# B&R Automation Studio project BottlePlant2 (part 2)

#### Main.st
```iecst
PROGRAM _INIT
	(* Insert code here *)
	gCamSequencer.Ctrl.MpAxisCamSequencer_0.Enable:=TRUE;
	gCamSequencer.Ctrl.MpAxisCamSequencer_1.Enable:=TRUE;
	gCamSequencer.State:=STATE_WORK_SEQUENCER;

	(* Zdefiniowanie podstawowych parametrów sequencera *)
	gCamSequencer.Ctrl.MpAxisCamSequencerPar_0.Deceleration:=1000;
	gCamSequencer.Ctrl.MpAxisCamSequencerPar_0.Configuration.Master:=ADR(gTranAxis);
	gCamSequencer.Ctrl.MpAxisCamSequencerPar_0.Configuration.StartState:=0;
	gCamSequencer.Ctrl.MpAxisCamSequencerPar_0.Configuration.State[0].Event[0].Type:=ncSIGNAL1;
	gCamSequencer.Ctrl.MpAxisCamSequencerPar_0.Configuration.State[0].Event[0].Attribute:=ncAT_ONCE;
	gCamSequencer.Ctrl.MpAxisCamSequencerPar_0.Configuration.State[0].Event[0].NextState:=1;

	gCamSequencer.Ctrl.MpAxisCamSequencerPar_0.Configuration.State[1].CompMode:=ncOFF;
	gCamSequencer.Ctrl.MpAxisCamSequencerPar_0.Configuration.State[1].CamProfileIndex:=16#ffff;
	gCamSequencer.Ctrl.MpAxisCamSequencerPar_0.Configuration.State[1].MasterCompDistance:=0;
	gCamSequencer.Ctrl.MpAxisCamSequencerPar_0.Configuration.State[1].SlaveCompDistance:=0;
	gCamSequencer.Ctrl.MpAxisCamSequencerPar_0.Configuration.State[1].MasterFactor:=400*100;
	gCamSequencer.Ctrl.MpAxisCamSequencerPar_0.Configuration.State[1].SlaveFactor:=400*100;
	gCamSequencer.Ctrl.MpAxisCamSequencerPar_0.Configuration.State[1].Event[0].Type:=ncST_END;
	gCamSequencer.Ctrl.MpAxisCamSequencerPar_0.Configuration.State[1].Event[0].Attribute:=ncST_END;
	gCamSequencer.Ctrl.MpAxisCamSequencerPar_0.Configuration.State[1].Event[0].NextState:=2;

	gCamSequencer.Ctrl.MpAxisCamSequencerPar_0.Configuration.State[2].CompMode:=ncOFF;
	gCamSequencer.Ctrl.MpAxisCamSequencerPar_0.Configuration.State[2].CamProfileIndex:=16#ffff;
	gCamSequencer.Ctrl.MpAxisCamSequencerPar_0.Configuration.State[2].MasterCompDistance:=0;
	gCamSequencer.Ctrl.MpAxisCamSequencerPar_0.Configuration.State[2].SlaveCompDistance:=0;
	gCamSequencer.Ctrl.MpAxisCamSequencerPar_0.Configuration.State[2].MasterFactor:=90*100;
	gCamSequencer.Ctrl.MpAxisCamSequencerPar_0.Configuration.State[2].SlaveFactor:=-400*100;
	gCamSequencer.Ctrl.MpAxisCamSequencerPar_0.Configuration.State[2].Event[0].Type:=ncST_END;
	gCamSequencer.Ctrl.MpAxisCamSequencerPar_0.Configuration.State[2].Event[0].Attribute:=ncST_END;
	gCamSequencer.Ctrl.MpAxisCamSequencerPar_0.Configuration.State[2].Event[0].NextState:=0;

	(* drugi seq *)
	gCamSequencer.Ctrl.MpAxisCamSequencerPar_1.Deceleration:=1000;
	gCamSequencer.Ctrl.MpAxisCamSequencerPar_1.Configuration.Master:=ADR(gCartAxis);
	gCamSequencer.Ctrl.MpAxisCamSequencerPar_1.Configuration.StartState:=0;
	gCamSequencer.Ctrl.MpAxisCamSequencerPar_1.Configuration.State[0].Event[0].Type:=ncSIGNAL1;
	gCamSequencer.Ctrl.MpAxisCamSequencerPar_1.Configuration.State[0].Event[0].Attribute:=ncAT_ONCE;
	gCamSequencer.Ctrl.MpAxisCamSequencerPar_1.Configuration.State[0].Event[0].NextState:=1;

	(* Nalewak inkrementalny -> nalewak idzie wraz z poziomem cieczy *)
	gCamSequencer.Ctrl.MpAxisCamSequencerPar_1.Configuration.State[1].CompMode:=ncOFF;
	gCamSequencer.Ctrl.MpAxisCamSequencerPar_1.Configuration.State[1].CamProfileIndex:=16#ffff;
	gCamSequencer.Ctrl.MpAxisCamSequencerPar_1.Configuration.State[1].MasterCompDistance:=0;
	gCamSequencer.Ctrl.MpAxisCamSequencerPar_1.Configuration.State[1].SlaveCompDistance:=0;
	gCamSequencer.Ctrl.MpAxisCamSequencerPar_1.Configuration.State[1].MasterFactor:=100*100;
	gCamSequencer.Ctrl.MpAxisCamSequencerPar_1.Configuration.State[1].SlaveFactor:=215*100;
	gCamSequencer.Ctrl.MpAxisCamSequencerPar_1.Configuration.State[1].Event[0].Type:=ncST_END;
	gCamSequencer.Ctrl.MpAxisCamSequencerPar_1.Configuration.State[1].Event[0].Attribute:=ncAT_ONCE;
	gCamSequencer.Ctrl.MpAxisCamSequencerPar_1.Configuration.State[1].Event[0].NextState:=2;

	gCamSequencer.Ctrl.MpAxisCamSequencerPar_1.Configuration.State[2].CompMode:=ncOFF;
	gCamSequencer.Ctrl.MpAxisCamSequencerPar_1.Configuration.State[2].CamProfileIndex:=16#ffff;
	gCamSequencer.Ctrl.MpAxisCamSequencerPar_1.Configuration.State[2].MasterCompDistance:=0;
	gCamSequencer.Ctrl.MpAxisCamSequencerPar_1.Configuration.State[2].SlaveCompDistance:=0;
	gCamSequencer.Ctrl.MpAxisCamSequencerPar_1.Configuration.State[2].MasterFactor:=215*100;
	gCamSequencer.Ctrl.MpAxisCamSequencerPar_1.Configuration.State[2].SlaveFactor:=-90*100;
	gCamSequencer.Ctrl.MpAxisCamSequencerPar_1.Configuration.State[2].Event[0].Type:=ncST_END;
	gCamSequencer.Ctrl.MpAxisCamSequencerPar_1.Configuration.State[2].Event[0].Attribute:=ncAT_ONCE;
	gCamSequencer.Ctrl.MpAxisCamSequencerPar_1.Configuration.State[2].Event[0].NextState:=3;

	gCamSequencer.Ctrl.MpAxisCamSequencerPar_1.Configuration.State[3].CompMode:=ncOFF;
	gCamSequencer.Ctrl.MpAxisCamSequencerPar_1.Configuration.State[3].CamProfileIndex:=16#ffff;
	gCamSequencer.Ctrl.MpAxisCamSequencerPar_1.Configuration.State[3].MasterCompDistance:=0;
	gCamSequencer.Ctrl.MpAxisCamSequencerPar_1.Configuration.State[3].SlaveCompDistance:=0;
	gCamSequencer.Ctrl.MpAxisCamSequencerPar_1.Configuration.State[3].MasterFactor:=54*100;
	gCamSequencer.Ctrl.MpAxisCamSequencerPar_1.Configuration.State[3].SlaveFactor:=-65*100;
	gCamSequencer.Ctrl.MpAxisCamSequencerPar_1.Configuration.State[3].Event[0].Type:=ncST_END;
	gCamSequencer.Ctrl.MpAxisCamSequencerPar_1.Configuration.State[3].Event[0].Attribute:=ncAT_ONCE;
	gCamSequencer.Ctrl.MpAxisCamSequencerPar_1.Configuration.State[3].Event[0].NextState:=4;

	gCamSequencer.Ctrl.MpAxisCamSequencerPar_1.Configuration.State[4].CompMode:=ncOFF;
	gCamSequencer.Ctrl.MpAxisCamSequencerPar_1.Configuration.State[4].CamProfileIndex:=16#ffff;
	gCamSequencer.Ctrl.MpAxisCamSequencerPar_1.Configuration.State[4].MasterCompDistance:=0;
	gCamSequencer.Ctrl.MpAxisCamSequencerPar_1.Configuration.State[4].SlaveCompDistance:=0;
	gCamSequencer.Ctrl.MpAxisCamSequencerPar_1.Configuration.State[4].MasterFactor:=22*100;
	gCamSequencer.Ctrl.MpAxisCamSequencerPar_1.Configuration.State[4].SlaveFactor:=-60*100;
	gCamSequencer.Ctrl.MpAxisCamSequencerPar_1.Configuration.State[4].Event[0].Type:=ncST_END;
	gCamSequencer.Ctrl.MpAxisCamSequencerPar_1.Configuration.State[4].Event[0].Attribute:=ncAT_ONCE;
	gCamSequencer.Ctrl.MpAxisCamSequencerPar_1.Configuration.State[4].Event[0].NextState:=0;

//	gCamSequencer.Ctrl.MpAxisCamSequencerPar_1.Configuration.State[1].CompMode:=ncOFF;
//	gCamSequencer.Ctrl.MpAxisCamSequencerPar_1.Configuration.State[1].CamProfileIndex:=16#ffff;
//	gCamSequencer.Ctrl.MpAxisCamSequencerPar_1.Configuration.State[1].MasterCompDistance:=0;
//	gCamSequencer.Ctrl.MpAxisCamSequencerPar_1.Configuration.State[1].SlaveCompDistance:=0;
//	gCamSequencer.Ctrl.MpAxisCamSequencerPar_1.Configuration.State[1].MasterFactor:=100*100;
//	gCamSequencer.Ctrl.MpAxisCamSequencerPar_1.Configuration.State[1].SlaveFactor:=215*100;
//	gCamSequencer.Ctrl.MpAxisCamSequencerPar_1.Configuration.State[1].Event[0].Type:=ncST_END;
//	gCamSequencer.Ctrl.MpAxisCamSequencerPar_1.Configuration.State[1].Event[0].Attribute:=ncAT_ONCE;
//	gCamSequencer.Ctrl.MpAxisCamSequencerPar_1.Configuration.State[1].Event[0].NextState:=2;
//
//	gCamSequencer.Ctrl.MpAxisCamSequencerPar_1.Configuration.State[2].CompMode:=ncOFF;
//	gCamSequencer.Ctrl.MpAxisCamSequencerPar_1.Configuration.State[2].CamProfileIndex:=16#ffff;
//	gCamSequencer.Ctrl.MpAxisCamSequencerPar_1.Configuration.State[2].MasterCompDistance:=0;
//	gCamSequencer.Ctrl.MpAxisCamSequencerPar_1.Configuration.State[2].SlaveCompDistance:=0;
//	gCamSequencer.Ctrl.MpAxisCamSequencerPar_1.Configuration.State[2].MasterFactor:=200*100;
//	gCamSequencer.Ctrl.MpAxisCamSequencerPar_1.Configuration.State[2].SlaveFactor:=0*100;
//	gCamSequencer.Ctrl.MpAxisCamSequencerPar_1.Configuration.State[2].Event[0].Type:=ncST_END;
//	gCamSequencer.Ctrl.MpAxisCamSequencerPar_1.Configuration.State[2].Event[0].Attribute:=ncAT_ONCE;
//	gCamSequencer.Ctrl.MpAxisCamSequencerPar_1.Configuration.State[2].Event[0].NextState:=3;
//
//	gCamSequencer.Ctrl.MpAxisCamSequencerPar_1.Configuration.State[3].CompMode:=ncOFF;
//	gCamSequencer.Ctrl.MpAxisCamSequencerPar_1.Configuration.State[3].CamProfileIndex:=16#ffff;
//	gCamSequencer.Ctrl.MpAxisCamSequencerPar_1.Configuration.State[3].MasterCompDistance:=0;
//	gCamSequencer.Ctrl.MpAxisCamSequencerPar_1.Configuration.State[3].SlaveCompDistance:=0;
//	gCamSequencer.Ctrl.MpAxisCamSequencerPar_1.Configuration.State[3].MasterFactor:=90*100;
//	gCamSequencer.Ctrl.MpAxisCamSequencerPar_1.Configuration.State[3].SlaveFactor:=-215*100;
//	gCamSequencer.Ctrl.MpAxisCamSequencerPar_1.Configuration.State[3].Event[0].Type:=ncST_END;
//	gCamSequencer.Ctrl.MpAxisCamSequencerPar_1.Configuration.State[3].Event[0].Attribute:=ncAT_ONCE;
//	gCamSequencer.Ctrl.MpAxisCamSequencerPar_1.Configuration.State[3].Event[0].NextState:=0;

END_PROGRAM

PROGRAM _CYCLIC
	(* Insert code here *)
	gCamSequencer.Ctrl.MpAxisCamSequencer_0.MpLink:=ADR(gCartAxisCfg);
	gCamSequencer.Ctrl.MpAxisCamSequencer_0.MpLinkMaster:=ADR(gTranAxisCfg);
	gCamSequencer.Ctrl.MpAxisCamSequencer_0.Parameters:=ADR(gCamSequencer.Ctrl.MpAxisCamSequencerPar_0);

	gCamSequencer.Ctrl.MpAxisCamSequencer_1.MpLink:=ADR(gPourAxisCfg);
	gCamSequencer.Ctrl.MpAxisCamSequencer_1.MpLinkMaster:=ADR(gCartAxisCfg);
	gCamSequencer.Ctrl.MpAxisCamSequencer_1.Parameters:=ADR(gCamSequencer.Ctrl.MpAxisCamSequencerPar_1);

	IF gCamSequencer.Ctrl.MpAxisCamSequencer_0.Error OR gCamSequencer.Ctrl.MpAxisCamSequencer_1.Error THEN
		gCamSequencer.State:=STATE_ERROR_SEQUENCER;
	END_IF;

	CASE gCamSequencer.State OF
		STATE_WORK_SEQUENCER:
			IF gCamSequencer.Ctrl.MpAxisCamSequencer_1.UpdateDone THEN
				gCamSequencer.Ctrl.MpAxisCamSequencer_1.Update:=FALSE;
			END_IF
			(* Warunek wzbudzający sygnał sequencera na 1 *)
			(* Jeśli zmienna licząca sygnał z czujnika butelek jest podzielna przez 5 oraz sygnał z tego czujnika ma zbocze opadające TO
			5 butelek jest pod nalewakami, zaczynamy sekwencję*)
			IF brmfmod(UDINT_TO_REAL(cntButelki),5.0)=0 AND EDGENEG(diButelka)THEN
				gCamSequencer.Ctrl.MpAxisCamSequencer_0.Signal1:=TRUE;
				gCamSequencer.Ctrl.MpAxisCamSequencer_1.Signal1:=TRUE;
			ELSE
				gCamSequencer.Ctrl.MpAxisCamSequencer_0.Signal1:=FALSE;
				gCamSequencer.Ctrl.MpAxisCamSequencer_1.Signal1:=FALSE;
			END_IF;

			IF gAxes.Ctrl.MpTransporterAxis.MoveActive AND (gCamSequencer.Ctrl.MpAxisCamSequencer_1.ActualStateIndex=2 OR gCamSequencer.Ctrl.MpAxisCamSequencer_1.ActualStateIndex=3) THEN
				DoPourer:=TRUE;
			ELSE
				DoPourer:=FALSE;
			END_IF
		STATE_ERROR_SEQUENCER:
			IF EDGEPOS(gCamSequencer.Cmd.ErrorReset) THEN
				gCamSequencer.Cmd.ErrorReset:=FALSE;
				gCamSequencer.Ctrl.MpAxisCamSequencer_0.ErrorReset:=TRUE;
				gCamSequencer.Ctrl.MpAxisCamSequencer_1.ErrorReset:=TRUE;
				//gCamSequencer.State:=STATE_WAIT_FOR_CMD_SEQUENCER;
			END_IF;
			IF NOT(gCamSequencer.Ctrl.MpAxisCamSequencer_0.Error) AND NOT(gCamSequencer.Ctrl.MpAxisCamSequencer_1.Error) THEN
				gCamSequencer.Ctrl.MpAxisCamSequencer_0.ErrorReset:=FALSE;
				gCamSequencer.Ctrl.MpAxisCamSequencer_1.ErrorReset:=FALSE;
	  			gCamSequencer.State:=STATE_WORK_SEQUENCER;
			END_IF;
	END_CASE;
	gCamSequencer.Ctrl.MpAxisCamSequencer_0();
	gCamSequencer.Ctrl.MpAxisCamSequencer_1();

END_PROGRAM

PROGRAM _EXIT
	(* Insert code here *)

END_PROGRAM
```

### UserCtrlGlobal.var
```iecst
VAR
	gCurrentUser : DINT;
END_VAR
```

### Program Logical/Software/Code/UserMgmt/UserCtrl

#### Types.typ
```iecst
TYPE
	UserCtrlType : STRUCT
		Login : MpUserLogin;
		LoginUI : MpUserLoginUI;
		UIConnect : MpUserLoginUIConnectType;
		UserData : UserDataType;

		UserManagerUI : MpUserManagerUI;
		UserManagerUISetup : MpUserMgrUISetupType;
		UserManagerUIConnect : MpUserMgrUIConnectType;

	END_STRUCT;

	UserDataType : STRUCT
		UserNameStr : STRING;
	END_STRUCT;

END_TYPE
```

#### Main.st
```iecst
PROGRAM _INIT
	(* Insert code here *)
	UserCtrl.Login.Enable:=TRUE;
	UserCtrl.LoginUI.Enable:=TRUE;
	UserCtrl.UserManagerUI.Enable:=TRUE;
END_PROGRAM

PROGRAM _CYCLIC
	(* Insert code here *)
	UserCtrl.Login.MpLink:=ADR(gUserLogin);
	UserCtrl.LoginUI.MpLink:=ADR(gUserLogin);
	UserCtrl.UserManagerUI.MpLink:=ADR(gUserLogin);

	UserCtrl.LoginUI.UIConnect:=ADR(UserCtrl.UIConnect);
	UserCtrl.UserManagerUI.UIConnect:=ADR(UserCtrl.UserManagerUIConnect);
	UserCtrl.UserManagerUI.UISetup:=UserCtrl.UserManagerUISetup;

	gCurrentUser:=UserCtrl.Login.CurrentLevel; // przekazanie lvl do głownego programu
	UserCtrl.Login.Logout:=gLogOutUser; //przekazanie z machineCtrl zmiennej która ustawia wylogowanie na TRUE
	UserCtrl.UserData.UserNameStr:=WSTRING_TO_STRING(UserCtrl.Login.CurrentUser);
	UserCtrl.Login();
	UserCtrl.LoginUI();
	UserCtrl.UserManagerUI();
END_PROGRAM

PROGRAM _EXIT
	(* Insert code here *)

END_PROGRAM
```

### Data object Logical/acp10etxen (Ett)

- acp10etxen.ett (not shown)

### Package Logical/gTranAxisobj - gTranAxisobj

### Data object Logical/gTranAxisobj/gTranAxisa (Apt)

#### gTranAxisa.apt
```
AcoposParameterTable:
  Root Parameters:
    110 = ncSWITCH_OFF (Name=CMD_SIMULATION)
```

### Data object Logical/gTranAxisobj/gTranAxisi (Ax)

#### gTranAxisi.ax
```
InitParameter (Version=5.12.2, NcSwId=Acp10)
  ACP10AXIS_typ:
    dig_in:
      level:
        reference = ncACTIV_HI
        pos_hw_end = ncACTIV_HI
        neg_hw_end = ncACTIV_HI
        trigger1 = ncACTIV_HI
        trigger2 = ncACTIV_HI
    encoder_if:
      parameter:
        count_dir = ncSTANDARD
        scaling:
          load:
            units = 1000
            rev_motor = 1
    limit:
      parameter:
        v_pos = 10000
        v_neg = 10000
        a1_pos = 50000
        a2_pos = 50000
        a1_neg = 50000
        a2_neg = 50000
        t_jolt = 0
        t_in_pos = 0
        pos_sw_end = 2000000000
        neg_sw_end = -2000000000
        ds_warning = 500
        ds_stop = 1000
        a_stop = 1.0e30
        dv_stop = 0
        dv_stop_mode = ncOFF
    controller:
      mode = ncPOSITION
      position:
        kv = 624.0
        tn = 0
        t_predict = 0.0004
        t_total = 0.0004
        p_max = 1.0e30
        i_max = 0
      speed:
        kv = 0.2
        tn = 0
        t_filter = 0.0
        isq_filter1:
          type = ncOFF
          a0 = 0.0
          a1 = 0.0
          b0 = 0.0
          b1 = 0.0
          b2 = 0.0
          c0_par_id = 0
          c1_par_id = 0
        isq_filter2:
          type = ncOFF
          a0 = 0.0
          a1 = 0.0
          b0 = 0.0
          b1 = 0.0
          b2 = 0.0
          c0_par_id = 0
          c1_par_id = 0
        isq_filter3:
          type = ncOFF
          a0 = 0.0
          a1 = 0.0
          b0 = 0.0
          b1 = 0.0
          b2 = 0.0
          c0_par_id = 0
          c1_par_id = 0
      uf:
        type = ncLINEAR + ncCORRECTION
        auto_config = ncMOTOR_PAR
        u0 = 0
        un = 0
        fn = 50.0
        k_f_slip = 0
      ff:
        mode = ncSTANDARD
        torque_load = 0.0
        torque_pos = 0.0
        torque_neg = 0.0
        kv_torque = 0.0
        inertia = 0.0
        t_filter_a = 0.0
      fb:
        mode = ncSTANDARD
        speed_mix_ratio = 0.0
        speed_kv = 2.0
      model:
        mass1:
          inertia = 0
          viscous_friction = 0
        mass2:
          inertia = 0
          viscous_friction = 0
          stiffness = 0
          damping = 0
    move:
      stop:
        parameter[0]:
          decel_ramp = ncA_LIMIT
          controller = ncON
        parameter[1]:
          decel_ramp = ncA_LIMIT
          controller = ncON
        parameter[2]:
          decel_ramp = ncA_LIMIT
          controller = ncON
        parameter[3]:
          decel_ramp = ncA_LIMIT
          controller = ncON
        quickstop:
          decel_ramp = ncA_LIMIT
          t_jolt = 0
        drive_error:
          decel_ramp = ncA_LIMIT
      homing:
        parameter:
          s = 0
          v_switch = 5000
          v_trigger = 500
          a = 50000
          mode = ncDIRECT
          edge_sw = ncPOSITIVE
          start_dir = ncPOSITIVE
          trigg_dir = ncPOSITIVE
          ref_pulse = ncOFF
          fix_dir = ncOFF
          tr_s_block = 0
          torque_lim = 0
          ds_block = 0
          ds_stop = 0
      basis:
        parameter:
          v_pos = 5000
          v_neg = 5000
          a1_pos = 50000
          a2_pos = 50000
          a1_neg = 50000
          a2_neg = 50000
    message:
      text:
        parameter:
          format = ncBREAK
          columns = 80
          data_modul = acp10etxen
```

### Package Logical/gCartAxisobj - gCartAxisobj

### Data object Logical/gCartAxisobj/gCartAxisa (Apt)

#### gCartAxisa.apt
```
AcoposParameterTable:
  Root Parameters:
    110 = ncSWITCH_ON (Name=CMD_SIMULATION)
```

### Data object Logical/gCartAxisobj/gCartAxisi (Ax)

#### gCartAxisi.ax
```
InitParameter (Version=5.12.2, NcSwId=Acp10)
  ACP10AXIS_typ:
    dig_in:
      level:
        reference = ncACTIV_HI
        pos_hw_end = ncACTIV_HI
        neg_hw_end = ncACTIV_HI
        trigger1 = ncACTIV_HI
        trigger2 = ncACTIV_HI
    encoder_if:
      parameter:
        count_dir = ncSTANDARD
        scaling:
          load:
            units = 1000
            rev_motor = 1
    limit:
      parameter:
        v_pos = 10000
        v_neg = 10000
        a1_pos = 50000
        a2_pos = 50000
        a1_neg = 50000
        a2_neg = 50000
        t_jolt = 0
        t_in_pos = 0
        pos_sw_end = 2000000000
        neg_sw_end = -2000000000
        ds_warning = 500
        ds_stop = 1000
        a_stop = 1.0e30
        dv_stop = 0
        dv_stop_mode = ncOFF
    controller:
      mode = ncPOSITION
      position:
        kv = 50
        tn = 0
        t_predict = 0.0004
        t_total = 0.0004
        p_max = 1.0e30
        i_max = 0
      speed:
        kv = 2.0
        tn = 0
        t_filter = 0.0
        isq_filter1:
          type = ncOFF
          a0 = 0.0
          a1 = 0.0
          b0 = 0.0
          b1 = 0.0
          b2 = 0.0
          c0_par_id = 0
          c1_par_id = 0
        isq_filter2:
          type = ncOFF
          a0 = 0.0
          a1 = 0.0
          b0 = 0.0
          b1 = 0.0
          b2 = 0.0
          c0_par_id = 0
          c1_par_id = 0
        isq_filter3:
          type = ncOFF
          a0 = 0.0
          a1 = 0.0
          b0 = 0.0
          b1 = 0.0
          b2 = 0.0
          c0_par_id = 0
          c1_par_id = 0
      uf:
        type = ncLINEAR + ncCORRECTION
        auto_config = ncMOTOR_PAR
        u0 = 0
        un = 0
        fn = 50.0
        k_f_slip = 0
      ff:
        mode = ncSTANDARD
        torque_load = 0.0
        torque_pos = 0.0
        torque_neg = 0.0
        kv_torque = 0.0
        inertia = 0.0
        t_filter_a = 0.0
      fb:
        mode = ncSTANDARD
        speed_mix_ratio = 0.0
        speed_kv = 2.0
      model:
        mass1:
          inertia = 0
          viscous_friction = 0
        mass2:
          inertia = 0
          viscous_friction = 0
          stiffness = 0
          damping = 0
    move:
      stop:
        parameter[0]:
          decel_ramp = ncA_LIMIT
          controller = ncON
        parameter[1]:
          decel_ramp = ncA_LIMIT
          controller = ncON
        parameter[2]:
          decel_ramp = ncA_LIMIT
          controller = ncON
        parameter[3]:
          decel_ramp = ncA_LIMIT
          controller = ncON
        quickstop:
          decel_ramp = ncA_LIMIT
          t_jolt = 0
        drive_error:
          decel_ramp = ncA_LIMIT
      homing:
        parameter:
          s = 0
          v_switch = 5000
          v_trigger = 500
          a = 50000
          mode = ncDIRECT
          edge_sw = ncPOSITIVE
          start_dir = ncPOSITIVE
          trigg_dir = ncPOSITIVE
          ref_pulse = ncOFF
          fix_dir = ncOFF
          tr_s_block = 0
          torque_lim = 0
          ds_block = 0
          ds_stop = 0
      basis:
        parameter:
          v_pos = 5000
          v_neg = 5000
          a1_pos = 50000
          a2_pos = 50000
          a1_neg = 50000
          a2_neg = 50000
    message:
      text:
        parameter:
          format = ncBREAK
          columns = 80
          data_modul = acp10etxen
```

### Package Logical/gPourAxisobj - gPourAxisobj

- Data object Logical/gPourAxisobj/gPourAxisa (Apt) (no source held here)

### Data object Logical/gPourAxisobj/gPourAxisi (Ax)

#### gPourAxisi.ax
```
InitParameter (Version=5.12.2, NcSwId=Acp10)
  ACP10AXIS_typ:
    dig_in:
      level:
        reference = ncACTIV_HI
        pos_hw_end = ncACTIV_HI
        neg_hw_end = ncACTIV_HI
        trigger1 = ncACTIV_HI
        trigger2 = ncACTIV_HI
    encoder_if:
      parameter:
        count_dir = ncSTANDARD
        scaling:
          load:
            units = 1000
            rev_motor = 1
    limit:
      parameter:
        v_pos = 10000
        v_neg = 10000
        a1_pos = 50000
        a2_pos = 50000
        a1_neg = 50000
        a2_neg = 50000
        t_jolt = 0
        t_in_pos = 0
        pos_sw_end = 2000000000
        neg_sw_end = -2000000000
        ds_warning = 500
        ds_stop = 1000
        a_stop = 1.0e30
        dv_stop = 0
        dv_stop_mode = ncOFF
    controller:
      mode = ncPOSITION
      position:
        kv = 619.0
        tn = 0
        t_predict = 0.0004
        t_total = 0.0004
        p_max = 1.0e30
        i_max = 0
      speed:
        kv = 0.15
        tn = 0
        t_filter = 0.0
        isq_filter1:
          type = ncOFF
          a0 = 0.0
          a1 = 0.0
          b0 = 0.0
          b1 = 0.0
          b2 = 0.0
          c0_par_id = 0
          c1_par_id = 0
        isq_filter2:
          type = ncOFF
          a0 = 0.0
          a1 = 0.0
          b0 = 0.0
          b1 = 0.0
          b2 = 0.0
          c0_par_id = 0
          c1_par_id = 0
        isq_filter3:
          type = ncOFF
          a0 = 0.0
          a1 = 0.0
          b0 = 0.0
          b1 = 0.0
          b2 = 0.0
          c0_par_id = 0
          c1_par_id = 0
      uf:
        type = ncLINEAR + ncCORRECTION
        auto_config = ncMOTOR_PAR
        u0 = 0
        un = 0
        fn = 50.0
        k_f_slip = 0
      ff:
        mode = ncSTANDARD
        torque_load = 0.0
        torque_pos = 0.0
        torque_neg = 0.0
        kv_torque = 0.0
        inertia = 0.0
        t_filter_a = 0.0
      fb:
        mode = ncSTANDARD
        speed_mix_ratio = 0.0
        speed_kv = 2.0
      model:
        mass1:
          inertia = 0
          viscous_friction = 0
        mass2:
          inertia = 0
          viscous_friction = 0
          stiffness = 0
          damping = 0
    move:
      stop:
        parameter[0]:
          decel_ramp = ncA_LIMIT
          controller = ncON
        parameter[1]:
          decel_ramp = ncA_LIMIT
          controller = ncON
        parameter[2]:
          decel_ramp = ncA_LIMIT
          controller = ncON
        parameter[3]:
          decel_ramp = ncA_LIMIT
          controller = ncON
        quickstop:
          decel_ramp = ncA_LIMIT
          t_jolt = 0
        drive_error:
          decel_ramp = ncA_LIMIT
      homing:
        parameter:
          s = 0
          v_switch = 5000
          v_trigger = 500
          a = 50000
          mode = ncDIRECT
          edge_sw = ncPOSITIVE
          start_dir = ncPOSITIVE
          trigg_dir = ncPOSITIVE
          ref_pulse = ncOFF
          fix_dir = ncOFF
          tr_s_block = 0
          torque_lim = 0
          ds_block = 0
          ds_stop = 0
      basis:
        parameter:
          v_pos = 5000
          v_neg = 5000
          a1_pos = 50000
          a2_pos = 50000
          a1_neg = 50000
          a2_neg = 50000
    message:
      text:
        parameter:
          format = ncBREAK
          columns = 80
          data_modul = acp10etxen
```

### GlobalRobVis.var - Global variables
```iecst
VAR
	diButelka : BOOL;
	AdrAxesPositions : UDINT;
	cntButelki : UDINT;
	posN : INT;
END_VAR
```

### GlobalRobVis.typ - Global data types
```iecst
TYPE
	AxesPositionsType : 	STRUCT
		Tasma : LREAL;
		Wozek : LREAL;
		Nalewak : LREAL;
	END_STRUCT;
END_TYPE
```

### Program Logical/Source/Misc/RobVis (IEC)

#### Main.st - Init, cyclic, exit code
```iecst
PROGRAM _INIT
	ModelConfig.Butelki.OffsetPierwszej := 7;
	ModelConfig.Butelki.Rozstaw := 100;
	ModelConfig.Butelki.Szerokosc := 80;

	ModelConfig.Wozek.OffsetWozka := 0;
END_PROGRAM

PROGRAM _CYCLIC

	IF AdrAxesPositions <> 0 THEN
		pAxesPositions ACCESS AdrAxesPositions;
	ELSE
		RETURN;
	END_IF
	TasmaPos1:=LREAL_TO_REAL(pAxesPositions.Tasma);
	TasmaPos1:=brmfmod(TasmaPos1,2300);

	// --------------------------------------------
	// Prepare correct positions for model
	// --------------------------------------------
	RobVisData.Tasma := ModelConfig.Butelki.OffsetPierwszej + TasmaPos1 + TasmaAxisPosition;
	RobVisData.Wozek := ModelConfig.Wozek.OffsetWozka + LREAL_TO_REAL(pAxesPositions.Wozek) + WozekAxisPosition;
	RobVisData.Nalewak := (LREAL_TO_REAL(pAxesPositions.Nalewak) + NalewakAxisPosition);
	RobVisData.SensorColor;

	// --------------------------------------------
	// Generator sygnalu czujnika butelki
	// --------------------------------------------
	FOR i := 0 TO 50 DO
		IF (RobVisData.Tasma > i*ModelConfig.Butelki.Rozstaw) AND (RobVisData.Tasma < (i*ModelConfig.Butelki.Rozstaw + ModelConfig.Butelki.Szerokosc)) THEN
			diButelka := TRUE;
			RobVisData.SensorColor := 5;
			EXIT;
		ELSE
			diButelka := FALSE;
			RobVisData.SensorColor := 11;
		END_IF
	END_FOR

	// --------------------------------------------
	// Licznik butelek
	// --------------------------------------------
	IF (diButelkaOld <> diButelka) AND diButelka THEN
		cntButelki := cntButelki + 1;
	END_IF
	diButelkaOld := diButelka;

	// --------------------------------------------
	// Tests
	// --------------------------------------------
	IF cmdTestModelMovements THEN
		TasmaAxisPosition := TasmaAxisPosition + 1;
		WozekAxisPosition := WozekAxisPosition + 1;
		NalewakAxisPosition := NalewakAxisPosition + 1;

		IF TasmaAxisPosition > 5000 THEN
			TasmaAxisPosition := 0;
		END_IF

		IF WozekAxisPosition > 1200 THEN
			WozekAxisPosition := 0;
		END_IF

		IF NalewakAxisPosition > 230 THEN
			NalewakAxisPosition := 0;
		END_IF
	END_IF

	// --------------------------------------------
	// Info: w tasku z napedami jest kod z przepisaniem pozycji napedow:

		// --------------------------------------------
		// Axes positions
		// --------------------------------------------
		// AdrAxesPositions := ADR(pAxesPositions);
		// AxesPositions.Tasma := MpAxisBasicList[0].Position;
		// AxesPositions.Wozek := MpAxisBasicList[1].Position;
		// AxesPositions.Nalewak := MpAxisBasicList[2].Position;

	// --------------------------------------------
	// --------------------------------------------

END_PROGRAM
```

#### Types.typ - Local data types
```iecst
TYPE
	ModelConfigButelkiType : 	STRUCT
		Rozstaw : REAL; (*Rozstaw - o ile butelki sa oddalone od siebie - od srodka do srodka butelki*)
		Szerokosc : REAL; (*Szerokosc butelki*)
		OffsetPierwszej : REAL; (*Pozycja kiedy pierwsza butelka jest rowno z poczatkiem stolu*)
	END_STRUCT;
	ModelConfigWozekType : 	STRUCT
		OffsetWozka : REAL; (*Pozycja kiedy wozek jest umieszczony dokladnie nad butelkami w pozycji zerowej*)
	END_STRUCT;
	ModelConfigType : 	STRUCT
		Butelki : ModelConfigButelkiType;
		Wozek : ModelConfigWozekType;
	END_STRUCT;
	RobVisPosType : 	STRUCT
		Tasma : REAL;
		Wozek : REAL;
		Nalewak : REAL;
		SensorColor : USINT;
	END_STRUCT;
END_TYPE
```

#### Variables.var - Local variables
```iecst
VAR
	cmdTestModelMovements : BOOL;
	RobVisData : RobVisPosType;
	ModelConfig : ModelConfigType;
	i : INT;
	diButelkaOld : BOOL;
	TasmaAxisPosition : REAL;
	WozekAxisPosition : REAL;
	NalewakAxisPosition : REAL;
	TasmaPos1 : REAL;
	TasmaPos2 : REAL;
	pAxesPositions : REFERENCE TO AxesPositionsType;
END_VAR
```
